	    80: //Error Reading Access
	        #Done := true;
	        #Busy := false;
	        #Error := TRUE;
	        #ErrorId := #st_StatusRead;
	        
	    90:  // Error while Write Access
	        #Done := true;
	        #Busy := false;
	        #Error := TRUE;
	        #ErrorId := #st_StatusWR;
	        
	        
	    100: // read successfully
	        #Done := true;
	        #Busy := false;
	        #Error := false;
	        
	    150:// write successfully
	        #Done := true;
	        #Busy := false;
	        #Error := false;
	        
	    200:  //Error while reading
	        #Done := true;
	        #Busy := false;
	        #Error := TRUE;
	        
	    300:  //Error while writing
	        #Done := true;
	        #Busy := false;
	        #Error := TRUE;
	        
	END_CASE;
	
	IF NOT #Enable THEN
	    #st_step := 0;
	    #st_ReqRef := 1;
	    #Done := false;
	    #Busy := false;
	    #Error := false;
	    #ErrorId := 16#00000000;
	    #ValueReadBOOL := false;
	    #ValueReadLINT := 0;
	    #ValueReadREAL := 0.0;
	    #st_StatusRead := 0;
	    #st_ErrorCounter := 0;
	END_IF;
END_FUNCTION_BLOCK

FUNCTION "Festo_Messages_Drives_EN" : Void
TITLE = Meldungen von CMMT MotorControllern
{ S7_Optimized_Access := 'TRUE' }
AUTHOR : LWNR
VERSION : 1.1
//Dieser Baustein gibt anhand der Meldungs-ID den Meldetext des Diagnose-
//ereignisses in Klartext (als STRING) aus.
//Weiterhin wird die Hauptgruppe, die Untergruppe, die Beschreibung sowie eine Abhilfe der anstehende Diasgnosemeldung in Klartext (als STRING) ausgegeben.
//Es sind alle Arten von Meldungen (Informationen, Warnungen und Fehler) der Geräte CMMT-AS und CMMT-ST enthalten.
   VAR_INPUT 
      ActFault_Drive : Word;   // Actual fault number of the drive
      ActWarning_Drive : Word;   // Actual warning number of the drive
   END_VAR

   VAR_OUTPUT 
      strMessage : String;   // Error or warning message
   END_VAR

   VAR_TEMP 
      MessageNo : Word;
   END_VAR


BEGIN
	(*############################################################
	    FESTO SE & Co. KG, Esslingen
	    Copyright (c) 2020. All rights reserved.    
	
	    NAME OF FUNCTION BLOCK:         Festo_Messages_Drives_EN
	    VERSION NUMBER:                 V1.1
	    COMPOSER:                       Festo
	    
	    -----------------------------------------------------
	   Date        Name                Activity                                                                              
	   20.02.2020  lwnr                created (V1.0)
	   09.12.2022  bkle                name changed 
	                                   Input: ActWarning_Drive added for warnings (V1.1)
	############################################################*)
	IF #ActFault_Drive <> 0 THEN
	    #MessageNo := #ActFault_Drive;
	ELSIF #ActWarning_Drive <> 0 THEN
	    #MessageNo := #ActWarning_Drive;
	END_IF;
	
	CASE WORD_TO_INT(#MessageNo) OF
	    0:
	        #strMessage := 'no error';
	        
	        (***************************************************************************)
	        (*                       Main group 1 - Current                             *)
	        (***************************************************************************)
	        
	        (* Subgroup 1 - Short circuit *)
	    10:
	        #strMessage := 'Short circuit motor phases/braking resistor';
	       
	    11:
	        #strMessage := 'Error on over-current monitoring';
	        
	        
	        (* Subgroup 2 - I²T *)
	    12:
	        #strMessage := 'I2t monitoring: motor warning limit';
	        
	    13:
	        #strMessage := 'I2t monitoring: motor error limit';
	        
	    14:
	        #strMessage := 'I2t monitoring: output stage warning limit';
	
	        
	    15:
	        #strMessage := 'I2t monitoring: output stage error limit';
	        
	    16:
	        #strMessage := 'I2t monitoring: output stage in standstill warning limit';
	        
	    17:
	        #strMessage := 'I2t monitoring: output stage in standstill error limit';
	        
	    18:
	        #strMessage := 'I2t monitoring motor: parameterisation invalid';
	        
	    258:
	        #strMessage := 'I2t monitoring: motor warning limit';
	        
	    259:
	        #strMessage := 'I2t monitoring: motor error limit';
	        
	        (* Subgroup 3 - braking resistor *)
	    19:
	        #strMessage := 'Warning: pulse energy monitoring, braking resistor';
	        
	    20:
	        #strMessage := 'Error: pulse energy monitoring, braking resistor';
	        
	    21:
	        #strMessage := 'Parameterisation of pulse energy monitoring for braking resistor invalid';
	        
	        
	        
	        (***************************************************************************)
	        (*                       Main group 2 - Voltage                          *)
	        (***************************************************************************)
	        
	        (* Subgroup 1 - Supply *)
	    22:
	        #strMessage := 'Undervoltage in logic supply (PS) 24 V DC';
	        
	    23:
	        #strMessage := 'Overvoltage in logic supply (PS) 24 V DC';
	        
	    24:
	        #strMessage := 'Undervoltage in logic supply 5V internal';
	        
	    25:
	        #strMessage := 'Overvoltage in logic supply 5V internal';
	        
	    26:
	        #strMessage := 'Undervoltage in logic supply 3.3V internal';
	        
	    27:
	        #strMessage := 'Overvoltage in logic supply 3.3V internal';
	        
	    28:
	        #strMessage := 'Undervoltage in logic supply safety section 3.3V internal';
	        
	    29:
	        #strMessage := 'Overvoltage in logic supply safety section 3.3V internal';
	        
	        
	        (* Subgroup 2 - intermediate circuit *)
	    30:
	        #strMessage := 'Overvoltage in intermediate circuit';
	        
	    31:
	        #strMessage := 'Undervoltage in intermediate circuit';
	        
	    32:
	        #strMessage := 'Intermediate circuit danger threshold reached';
	        
	    33:
	        #strMessage := 'DC link voltage too low following power failure';
	        
	    34:
	        #strMessage := 'Intermediate circuit precharge time exceeded';
	        
	    35:
	        #strMessage := 'Residual voltage too high following rapid discharge';
	        
	    286:
	        #strMessage := 'The DC relay for loading the DC link does not open';
	        
	    287:
	        #strMessage := 'The DC relay for charging the DC link does not close';
	        
	        
	        (* Subgroup 3 - Mains volatge *)
	    36:
	        #strMessage := 'No mains voltage';
	        
	    37:
	        #strMessage := 'System voltage dip detected';
	        
	    38:
	        #strMessage := 'Undervoltage in power supply';
	        
	    39:
	        #strMessage := 'Overvoltage in power supply';
	        
	    40:
	        #strMessage := 'Phase failure in power supply';
	        
	    41:
	        #strMessage := 'Powersupply signal shape NOT as configured';
	        
	    251:
	        #strMessage := 'Deactivation threshold for energy recovery reached';
	        
	        
	        
	        (* Subgroup 4 - Encoder supply voltage *)
	    42:
	        #strMessage := 'Supply voltage for encoder is outside monitoring thresholds';
	        
	    43:
	        #strMessage := 'Encoder supply voltage control failed';
	        
	        
	        (***************************************************************************)
	        (*                     Main group 3 - TEMPERATURE                          *)
	        (***************************************************************************)
	        
	        (* Subgroup 1 - GERAET *)
	    44:
	        #strMessage := 'Warning threshold: Insufficient temperature in device';
	        
	    45:
	        #strMessage := 'Insufficient temperature in device';
	        
	    46:
	        #strMessage := 'Warning threshold: Device overtemperature';
	        
	    47:
	        #strMessage := 'Device overtemperature';
	        
	        
	        (* Subgroup 2 - Output stage *)
	    48:
	        #strMessage := 'Warning threshold: Insufficient temperature in power section';
	        
	    49:
	        #strMessage := 'Insufficient temperature in output stage';
	        
	    50:
	        #strMessage := 'Warning threshold: Power section overtemperature';
	        
	    51:
	        #strMessage := 'Power section overtemperature';
	        
	        
	        (* Subgroup 3 - MOTOR *)
	    52:
	        #strMessage := 'Warning threshold: Insufficient temperature in motor';
	        
	    53:
	        #strMessage := 'Insufficient temperature in motor';
	        
	    54:
	        #strMessage := 'Warning threshold: Motor overtemperature';
	        
	    55:
	        #strMessage := 'Motor overtemperature';
	        
	        
	        (***************************************************************************)
	        (*                       Main group 5 - Motion                          *)
	        (***************************************************************************)
	        
	        (* Subgroup 1 - Homing *)
	    56:
	        #strMessage := 'Parameterisation of homing run invalid';
	        
	    57:
	        #strMessage := 'Homing: Timeout';
	        
	    58:
	        #strMessage := 'Homing: Search path exceeded';
	        
	        
	        (* Subgroup 2 - Movement calculation *)
	    59:
	        #strMessage := 'Task invalid';
	        
	    60:
	        #strMessage := 'Unknown motion task pending';
	        
	    61:
	        #strMessage := 'Task could not be executed as the drive control is missing';
	        
	    62:
	        #strMessage := 'Task could not be executed as a safety function is requested';
	        
	    63:
	        #strMessage := 'Calculation of brake travel failed';
	        
	    64:
	        #strMessage := 'Task could not be executed as no DC link voltage is present';
	        
	    65:
	        #strMessage := 'Motion task rejected in current status';
	        
	    66:
	        #strMessage := 'Task could not be executed as the encoder is not ready';
	        
	    67:
	        #strMessage := 'Task could not be executed as the drive is not referenced';
	        
	    68:
	        #strMessage := 'Task could not be executed as a reinitialization is required due to a parameter change';
	        
	    69:
	        #strMessage := 'Task could not be executed as a restart is required due to a parameter change';
	        
	    71:
	        #strMessage := 'An error occurred in the trajectory generator when calculating a movement profile';
	        
	    72:
	        #strMessage := 'The position specified for the trajectory generator is invalid';
	        
	    73:
	        #strMessage := 'The speed specified for the trajectory generator is invalid';
	        
	    74:
	        #strMessage := 'The acceleration specified for the trajectory generator is invalid';
	        
	    75:
	        #strMessage := 'The delay specified for the trajectory generator is invalid';
	        
	    76:
	        #strMessage := 'The jerk specified for the trajectory generator is invalid';
	        
	    77:
	        #strMessage := 'An error occurred in the trajectory generator when calculating a movement profile';
	        
	    78:
	        #strMessage := 'Stop ramp: Timeout';
	        
	    79:
	        #strMessage := 'The torque increase is invalid';
	        
	    80:
	        #strMessage := 'Simultaneous negative/positive directional lock';
	        
	    245:
	        #strMessage := 'Received PDO outside tolerance window';
	        
	    278:
	        #strMessage := 'Order could not be executed because a directional lock is active';
	        
	    279:
	        #strMessage := 'Fixed stop not reached';
	        
	    280:
	        #strMessage := 'Monitoring window exit fixed stop';
	        
	    364:
	        #strMessage := 'The preset profile velocity is 0';
	        
	        (***************************************************************************)
	        (*             Main group 6 - KONFIGURATION                *)
	        (***************************************************************************)
	        
	        (* Subgroup 0 - no categorie *)
	    70:
	        #strMessage := 'Record table parameter is invalid';
	        
	    81:
	        #strMessage := 'The operating mode of the regulator (position, speed, force, stop) does not match the parameterisation';
	        
	    82:
	        #strMessage := 'The parameterisation of the notch filter frequency is invalid';
	        
	    83:
	        #strMessage := 'Record table incorrect';
	        
	    84:
	        #strMessage := 'Parameterisation of switching frequency invalid';
	        
	    85:
	        #strMessage := 'The configuration of the digital inputs or outputs is invalid';
	        
	    248:
	        #strMessage := 'The parameterized motor type (servo, stepper, ...) is not supported';
	        
	    252:
	        #strMessage := 'Start and end voltage for reactive current braking incompatible';
	        
	    313:
	        #strMessage := 'Selection data trigger in function Variable signalling function invalid';
	        
	        
	        (* Subgroup 2 - Boundary value *)
	    86:
	        #strMessage := 'Setpoint torque and speed limit do not match';
	        
	    87:
	        #strMessage := 'Speed control limitation invalid';
	        
	    88:
	        #strMessage := 'Torque control limitation invalid';
	        
	    89:
	        #strMessage := 'Current control limitation invalid';
	        
	    90:
	        #strMessage := 'Maximum peak current control limitation invalid';
	        
	    91:
	        #strMessage := 'Parameterisation of nominal current/maximum peak current of motor invalid';
	        
	    273:
	        #strMessage := 'Change of control mode not permitted';
	        
	    274:
	        #strMessage := 'Movement order not permitted in controlled operation';
	        
	    275:
	        #strMessage := 'Change to close-loop operation not permitted';
	        
	        
	        (* Subgroup 5 - Parameter set *)
	    97:
	        #strMessage := 'Parameter set not found';
	        
	    98:
	        #strMessage := 'Parameter set invalid';
	        
	    99:
	        #strMessage := 'Parameter set incompatible';
	        
	    100:
	        #strMessage := 'Parameter not found';
	        
	    101:
	        #strMessage := 'Parameter not writable';
	        
	    102:
	        #strMessage := 'Transmission error in parameter set';
	        
	    103:
	        #strMessage := 'Parameter set: store failed';
	        
	    104:
	        #strMessage := 'Parameter set: delete failed';
	        
	    105:
	        #strMessage := 'Factory parameter not found';
	        
	    106:
	        #strMessage := 'Factory parameter set invalid';
	        
	    107:
	        #strMessage := 'Factory parameter set not found';
	        
	    108:
	        #strMessage := 'Factory parameter set incompatible';
	        
	    290:
	        #strMessage := 'Parameter set version older';
	        
	    291:
	        #strMessage := 'Parameter set version newer';
	        
	        
	        (***************************************************************************)
	        (*                        Main group 7 - Monitoring                      *)
	        (***************************************************************************)
	        
	        (* Subgroup 1 - Limits *)
	    109:
	        #strMessage := 'Negative software end position';
	        
	    110:
	        #strMessage := 'Positive software end position';
	        
	    111:
	        #strMessage := 'Limitation negative direction';
	        
	    112:
	        #strMessage := 'Limitation positive direction';
	        
	    113:
	        #strMessage := 'Parameterisation of software end positions';
	        
	    114:
	        #strMessage := 'Negative hardware limit switch reached';
	        
	    115:
	        #strMessage := 'Positive hardware limit switch reached';
	        
	    116:
	        #strMessage := 'Limitation by negative hardware limit switch';
	        
	    117:
	        #strMessage := 'Limitation by positive hardware limit switch';
	        
	    118:
	        #strMessage := 'Error: both hardware limit switches occupied';
	        
	    119:
	        #strMessage := 'Negative stroke limit reached';
	        
	    120:
	        #strMessage := 'Positive stroke limit reached';
	        
	        
	        (* Subgroup 2 - Motion monitoring *)
	    121:
	        #strMessage := 'Target position reached';
	        
	    122:
	        #strMessage := 'Target speed reached';
	        
	    123:
	        #strMessage := 'Target torque reached';
	        
	    124:
	        #strMessage := 'Standstill reached';
	        
	    125:
	        #strMessage := 'Standstill reached and within standstill window';
	        
	    126:
	        #strMessage := 'Position error: following error';
	        
	    127:
	        #strMessage := 'velocity: following error';
	        
	    128:
	        #strMessage := 'velocity monitoring reports velocity too high';
	        
	    129:
	        #strMessage := 'Drive has left the target range';
	        
	    130:
	        #strMessage := 'Reverse feed monitoring reports error';
	        
	    131:
	        #strMessage := 'Residual distance too low';
	        
	    132:
	        #strMessage := 'Trajectory completed setpoint value reached';
	        
	    133:
	        #strMessage := 'Position difference encoder 1 to encoder 2 too large';
	        
	        
	        (* Subgroup 3 - boundary values *)
	    134:
	        #strMessage := 'Voltage limiting active';
	        
	    135:
	        #strMessage := 'A limit for the speed or current is active';
	        
	        
	        (* Subgroup 4 - Zero angle *)
	    136:
	        #strMessage := 'Zero-angle location failed';
	        
	    137:
	        #strMessage := 'Commutation finding error';
	        
	        
	        (* Subgroup 5 - analog input *)
	    138:
	        #strMessage := 'Analogue setpoint specification limit exceeded';
	        
	        
	        
	        (***************************************************************************)
	        (*                      Main group 8 - Communication                       *)
	        (***************************************************************************)
	        
	        (* Subgroup 0 - no categorie *)
	    139:
	        #strMessage := 'Fieldbus not supported';
	        
	    140:
	        #strMessage := 'Failure of fieldbus synchronisation signal';
	        
	    243:
	        #strMessage := 'Invalid cycle time';
	        
	        
	        (* Subgroup 3 - PROFINET *)
	    141:
	        #strMessage := 'Invalid process data';
	        
	    373:
	        #strMessage := 'Failure of communication processor synchronisation';
	        
	        
	        (* Subgroup 9 - PROFIDRIVE *)
	    144:
	        #strMessage := 'Application class not supported';
	        
	    145:
	        #strMessage := 'Telegram not supported';
	        
	    288:
	        #strMessage := 'ProfiDrive test fault 1';
	        
	    289:
	        #strMessage := 'ProfiDrive test fault 2';
	        
	    294:
	        #strMessage := 'PLC Control Bit is not set';
	        
	    299:
	        #strMessage := 'clock cycle synchronous operation sign-of-life failure';
	        
	    382:
	        #strMessage := 'Invalid configuration Extended process data';
	        
	        
	        (* Subgroup 12 - others *)
	    250:
	        #strMessage := 'Invalid operating mode';
	        
	    272:
	        #strMessage := 'Resolution position factor group invalid';
	        
	        
	        (***************************************************************************)
	        (*                     Main group 9 - Safety                               *)
	        (***************************************************************************)
	        
	        (* Subgroup 0 - no categorie *)
	    146:
	        #strMessage := 'Safety function requested';
	        
	    147:
	        #strMessage := 'Plausibility check of safety feedback signals';
	        
	        
	        (* Subgroup 1 - STO *)
	    148:
	        #strMessage := 'STO: Discrepancy time exceeded';
	        
	    149:
	        #strMessage := 'Plausibility check #STO-A/B';
	        
	    150:
	        #strMessage := 'Sequence monitoring #STO-A/B';
	        
	        
	        (* Subgroup 2 - SBC *)
	    151:
	        #strMessage := 'Plausibility check #SBC-A/B';
	        
	    152:
	        #strMessage := 'SBC: Discrepancy time exceeded';
	        
	        
	        (***************************************************************************)
	        (*                     Main group 10 - Internal hardware                   *)
	        (***************************************************************************)
	        
	        (* Subgroup 1 - Module error *)
	    153:
	        #strMessage := 'RTE module cannot be reached';
	        
	    154:
	        #strMessage := 'Internalisation of RTE module failed';
	        
	    155:
	        #strMessage := 'Error: fan faulty';
	        
	    156:
	        #strMessage := 'Common error power output stage';
	        
	    157:
	        #strMessage := 'FPGA does not start up';
	        
	    158:
	        #strMessage := 'FPGA version invalid';
	        
	    199:
	        #strMessage := 'Synchronisation with FPGA failed';
	        
	    249:
	        #strMessage := 'Error RTE module watchdog monitoring';
	        
	        
	        
	        (***************************************************************************)
	        (*                         Main group 11 - SOFTWARE                       *)
	        (***************************************************************************)
	        
	        (* Subgroup 1 - EXCEPTION *)
	        
	    159:
	        #strMessage := 'Data directory memory full';
	        
	    160:
	        #strMessage := 'Data directory indexed twice';
	        
	    161:
	        #strMessage := 'Overflow diagnostic register';
	        
	    162:
	        #strMessage := 'Overflow diagnostic register buffer';
	        
	    163:
	        #strMessage := 'Error user unit conversion';
	        
	    244:
	        #strMessage := 'Undervoltage RTE module';
	        
	        
	        (* Subgroup 2 - TASK *)
	    164:
	        #strMessage := 'Process runtime exceeded';
	        
	    165:
	        #strMessage := 'Timeout process level 0';
	        
	    166:
	        #strMessage := 'Timeout process level 1';
	        
	    167:
	        #strMessage := 'Timeout process level 2';
	        
	    168:
	        #strMessage := 'Timeout process level 3';
	        
	    169:
	        #strMessage := 'Timeout process level 4';
	        
	    170:
	        #strMessage := 'Timeout process level 5';
	        
	    171:
	        #strMessage := 'Timeout process level 6';
	        
	    172:
	        #strMessage := 'Timeout process level 7';
	        
	        
	        (* Subgroup 3 - File system *)
	    173:
	        #strMessage := 'File system faulty';
	        
	    174:
	        #strMessage := 'File: user file (backup) invalid';
	        
	    175:
	        #strMessage := 'Creation of user file (backup) not possible';
	        
	    176:
	        #strMessage := 'CRC error in user file';
	        
	    177:
	        #strMessage := 'File: user file invalid';
	        
	    178:
	        #strMessage := 'New user file has been created';
	        
	    179:
	        #strMessage := 'Writing to user file not possible';
	        
	    180:
	        #strMessage := 'Unknown user file error';
	        
	        
	        (* Subgroup 4 - FIRMWAREUPDATE *)
	    181:
	        #strMessage := 'Writing to firmware failed';
	        
	    182:
	        #strMessage := 'Reading from firmware failed';
	        
	    183:
	        #strMessage := 'Firmware invalid';
	        
	    184:
	        #strMessage := 'Firmware incompatible';
	        
	    185:
	        #strMessage := 'Firmware save location invalid';
	        
	    186:
	        #strMessage := 'Firmware save location empty';
	        
	    187:
	        #strMessage := 'Firmware update not allowed';
	        
	    188:
	        #strMessage := 'Firmware package in use';
	        
	    189:
	        #strMessage := 'System error during firmware update';
	        
	    190:
	        #strMessage := 'Firmware update failed';
	        
	        
	        (* Subgroup 5 - Device configuration *)
	    191:
	        #strMessage := 'Calibration data incorrect: Safety';
	        
	    192:
	        #strMessage := 'Device data incorrect';
	        
	    193:
	        #strMessage := 'Device data incorrect: control section';
	        
	    194:
	        #strMessage := 'Device data incorrect: communication section';
	        
	    195:
	        #strMessage := 'Device data incorrect: Safety';
	        
	    196:
	        #strMessage := 'Calibration data incorrect: control section';
	        
	    197:
	        #strMessage := 'Calibration data incorrect: power section';
	        
	    198:
	        #strMessage := 'Device data incorrect: power section';
	        
	    200:
	        #strMessage := 'Current sensor calibration invalid';
	        
	    201:
	        #strMessage := 'Device not configured';
	        
	    202:
	        #strMessage := 'Device data: store failed';
	        
	        
	        (* Subgroup 6 - LIBRTE *)
	    203:
	        #strMessage := 'Answer to a read request missing in LibRTE';
	        
	    285:
	        #strMessage := 'Error communication module mailbox';
	        
	    300:
	        #strMessage := 'COM module error';
	        
	        
	        (* Subgroup 7 - WARMSTART *)
	    204:
	        #strMessage := 'Initialization failed';
	        
	    205:
	        #strMessage := 'Task ignored as reinitialization not possible';
	        
	    271:
	        #strMessage := 'Reinitialization failed';
	        
	        
	        (* Subgroup 8 - version  management *)
	    206:
	        #strMessage := 'Hardware does not correspond to expected revision status';
	        
	    207:
	        #strMessage := 'Hardware does not correspond to expected compatibility state';
	        
	        
	        
	        (***************************************************************************)
	        (*                         Main group 12 - maintenance                        *)
	        (***************************************************************************)
	        
	        (* Subgroup 1 - Mileage *)
	    208:
	        #strMessage := 'Maximum value for the mileage is reached';
	        
	    209:
	        #strMessage := 'Mileage danger threshold reached';
	        
	    210:
	        #strMessage := 'Mileage error threshold reached';
	        
	    211:
	        #strMessage := 'Maximum load change value reached';
	        
	    212:
	        #strMessage := 'Load change danger threshold reached';
	        
	    213:
	        #strMessage := 'Load change error threshold reached';
	        
	        
	        
	        (***************************************************************************)
	        (*                      Main group 13 - Others                     *)
	        (***************************************************************************)
	        
	        (* Subgroup 1 - diagnosis *)
	    214:
	        #strMessage := 'Message acknowledgment';
	        
	    215:
	        #strMessage := 'Diagnostics log file has invalid format';
	        
	    216:
	        #strMessage := 'Loss of messages from diagnostics log';
	        
	        
	        (* Subgroup 2 - AUTOTUNING *)
	    217:
	        #strMessage := 'Autotuning aborted';
	        
	    218:
	        #strMessage := 'Autotuning travel insufficient';
	        
	    219:
	        #strMessage := 'Autotuning controller parameters invalid';
	        
	    220:
	        #strMessage := 'Transmission of autotuning measured values failed';
	        
	        
	        
	        
	        
	        
	        (***************************************************************************)
	        (*                     Main group 16 - External device                     *)
	        (***************************************************************************)
	        
	        (* Subgroup 1 - CDSB *)
	    221:
	        #strMessage := 'CDSB display file faulty';
	        
	    222:
	        #strMessage := 'JSON display description for CDSB too large';
	        
	    223:
	        #strMessage := 'SPI communication too slow';
	        
	        
	        
	        
	        
	        (***************************************************************************)
	        (*                   Main group 17 - Safety (data)                         *)
	        (***************************************************************************)
	        
	        (* Subgroup 1 - User login *)
	    224..225:
	        #strMessage := 'Login completed';
	        
	    226:
	        #strMessage := 'Login error';
	        
	        
	        
	        
	        
	        (***************************************************************************)
	        (*                        Main group 18 - Encoder                          *)
	        (***************************************************************************)
	        
	        (* Subgroup 0 - no cetegorie *)
	    92:
	        #strMessage := 'Motor change detected, commutation angle invalid';
	        
	    93:
	        #strMessage := 'Motor change detected, zero point offset invalid';
	        
	    94:
	        #strMessage := 'Commutation angle in encoder invalid';
	        
	    95:
	        #strMessage := 'Encoder type plate invalid';
	        
	    96:
	        #strMessage := 'Encoder type plate (user-defined) invalid';
	        
	    227:
	        #strMessage := 'Encoder identification reports incorrect encoder type';
	        
	    318:
	        #strMessage := 'State transition error';
	        
	        
	        (* Subgroup 1 - ENDAT*)
	    228:
	        #strMessage := 'Common error EnDat 2.1';
	        
	    229:
	        #strMessage := 'Common error EnDat 2.2';
	        
	        
	        (* Subgroup 2 - HYPERFACE*)
	    230:
	        #strMessage := 'Vector length invalid';
	        
	    231:
	        #strMessage := 'Quadrant invalid';
	        
	    232:
	        #strMessage := 'Hiperface communication timeout';
	        
	    233:
	        #strMessage := 'Error in CRC protocol Hiperface';
	        
	    234:
	        #strMessage := 'Common error Hiperface';
	        
	    276:
	        #strMessage := 'Quadrant unstable';
	        
	        
	        (* Subgroup 3 - QUADRATURE (incremental encoder)*)
	    235:
	        #strMessage := 'Incremental encoder analysis invalid';
	        
	    301:
	        #strMessage := 'Increments between Z-pulses invalid';
	        
	        
	        (* Subgroup 4 - NIKON A*)
	    236:
	        #strMessage := 'Protocol error Nikon-A encoder';
	        
	    237:
	        #strMessage := 'Timeout Nikon-A encoder';
	        
	    238:
	        #strMessage := 'CRC error Nikon-A encoder';
	        
	        
	        (* Subgroup 5 - BISS C*)
	    239:
	        #strMessage := 'BISSC encoder analysis invalid';
	        
	        
	        (* Subgroup 6 - SIN/COS*)
	    240:
	        #strMessage := 'Vector length invalid';
	        
	    241:
	        #strMessage := 'Quadrant invalid';
	        
	    242:
	        #strMessage := 'Timeout Geberinitialisierung';
	        
	    277:
	        #strMessage := 'Error SIN/COS-encoder';
	        
	        
	        (* Subgroup 7 - encoder systems *)
	    365:
	        #strMessage := 'Invalid request Gn_STW1.4...7';
	        
	    366:
	        #strMessage := 'Function not supported Gn_STW1';
	        
	    367:
	        #strMessage := 'Axis parking not possible';
	        
	    368:
	        #strMessage := 'Error reference marks search';
	        
	    369:
	        #strMessage := 'Error Read Position Reference mark';
	        
	    370:
	        #strMessage := 'Error measuring on the fly';
	        
	    371:
	        #strMessage := 'Error Read Position Measure on the fly';
	        
	    372:
	        #strMessage := 'Error Transfer absolute position to Gn_XIST2';
	        
	    ELSE  // Statement section ELSE
	        #strMessage := 'unknown';
	END_CASE;
	
END_FUNCTION

FUNCTION_BLOCK "LK_G5000"   // FB6, LAD
{ S7_Optimized_Access := 'TRUE' }
VERSION : 0.1
// stored: AutoNumber true, IsIECCheckEnabled false, IsRetainMemResEnabled false, MemoryReserve 100, SetENOAutomatically false, UDAEnableTagReadback false
BEGIN

REGION Network 1: Write / Read data in and from DB - CTRL_ BITS
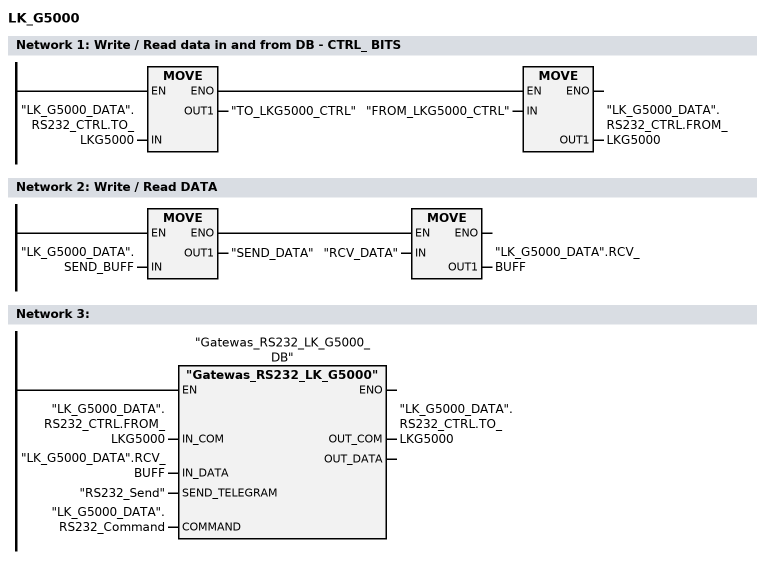
   RUNG wire#powerrail
      Move(in := "LK_G5000_DATA".RS232_CTRL.TO_LKG5000, out1 => "TO_LKG5000_CTRL")
      Move(in := "FROM_LKG5000_CTRL", out1 => "LK_G5000_DATA".RS232_CTRL.FROM_LKG5000)
   END_RUNG
   // the same network as SCL:
   "TO_LKG5000_CTRL" := "LK_G5000_DATA".RS232_CTRL.TO_LKG5000;
   "LK_G5000_DATA".RS232_CTRL.FROM_LKG5000 := "FROM_LKG5000_CTRL";
END_REGION

REGION Network 2: Write / Read DATA
   RUNG wire#powerrail
      Move(in := "LK_G5000_DATA".SEND_BUFF, out1 => "SEND_DATA")
      Move(in := "RCV_DATA", out1 => "LK_G5000_DATA".RCV_BUFF)
   END_RUNG
   // the same network as SCL:
   "SEND_DATA" := "LK_G5000_DATA".SEND_BUFF;
   "LK_G5000_DATA".RCV_BUFF := "RCV_DATA";
END_REGION

REGION Network 3
   RUNG wire#powerrail
      "Gatewas_RS232_LK_G5000_DB"(IN_COM := "LK_G5000_DATA".RS232_CTRL.FROM_LKG5000, IN_DATA := "LK_G5000_DATA".RCV_BUFF, SEND_TELEGRAM := "RS232_Send", COMMAND := "LK_G5000_DATA".RS232_Command, OUT_COM => "LK_G5000_DATA".RS232_CTRL.TO_LKG5000, OUT_DATA =>)
   END_RUNG
   // the same network as SCL:
   "Gatewas_RS232_LK_G5000_DB"(IN_COM := "LK_G5000_DATA".RS232_CTRL.FROM_LKG5000,   // "Gatewas_RS232_LK_G5000"
                           IN_DATA := "LK_G5000_DATA".RCV_BUFF,
                           SEND_TELEGRAM := "RS232_Send",
                           COMMAND := "LK_G5000_DATA".RS232_Command,
                           OUT_COM => "LK_G5000_DATA".RS232_CTRL.TO_LKG5000);
END_REGION
END_FUNCTION_BLOCK

FUNCTION_BLOCK "Gatewas_RS232_LK_G5000"   // FB10, LAD
{ S7_Optimized_Access := 'TRUE' }
VERSION : 0.1
// stored: AutoNumber true, IsIECCheckEnabled false, IsRetainMemResEnabled false, MemoryReserve 100, SetENOAutomatically false, UDAEnableTagReadback false
   VAR_INPUT
      IN_COM : "UDT_LKG5000_RS232_RCV";
      IN_DATA : "UDT_RS232_RCV_DATA";
      SEND_TELEGRAM : Bool;
      COMMAND : String[10];
   END_VAR
   VAR_OUTPUT
      OUT_COM : "UDT_LKG5000_RS232_SEND";
      OUT_DATA : "UDT_RS232_SEND_DATA";
   END_VAR
   VAR
      COMMAND_SIGN : Array[0..10] of Char;
      Cnt_Command : UInt;
      IEC_Timer_0_Instance { S7_SetPoint := 'True'} : TOF_TIME;
      IEC_Timer_0_Instance_1 { S7_SetPoint := 'True'} : TOF_TIME;
   END_VAR
BEGIN

REGION Network 2 (SCL)
   Strg_TO_Chars(Strg:=#COMMAND,
                 pChars:=0,
                 Cnt=>#Cnt_Command,
                 Chars:=#COMMAND_SIGN);





   // Send frame
   #OUT_COM.Sendframe_size := 20;
   // Receive Frame
   #OUT_COM.Recvframe_size := 20;


   //#OUT_DATA.Data[0] := B#16#02;
   #OUT_DATA.Data[0] := #COMMAND_SIGN[0];
   #OUT_DATA.Data[1] := #COMMAND_SIGN[1];
   #OUT_DATA.Data[2] := #COMMAND_SIGN[2];
   #OUT_DATA.Data[3] := #COMMAND_SIGN[3];
   #OUT_DATA.Data[4] := #COMMAND_SIGN[4];
   #OUT_DATA.Data[5] :=  B#16#D0;

   //#OUT_DATA.Data[5] := #COMMAND_SIGN[5];
   //#OUT_DATA.Data[6] := #COMMAND_SIGN[6];
   //#OUT_DATA.Data[7] := #COMMAND_SIGN[7];
   //#OUT_DATA.Data[8] := #COMMAND_SIGN[8];
   //#OUT_DATA.Data[9] := #COMMAND_SIGN[9];
   //#OUT_DATA.Data[10] := #COMMAND_SIGN[10];
   //#OUT_DATA.Data[11] := #COMMAND_SIGN[11];
   //#OUT_DATA.Data[12] := #COMMAND_SIGN[12];
   //#OUT_DATA.Data[13] := #COMMAND_SIGN[13];
   //#OUT_DATA.Data[14] := #COMMAND_SIGN[14];
   //#OUT_DATA.Data[15] := #COMMAND_SIGN[15];
   //#OUT_DATA.Data[16] := #COMMAND_SIGN[16];
   //#OUT_DATA.Data[17] := #COMMAND_SIGN[17];
   //#OUT_DATA.Data[18] := #COMMAND_SIGN[18];
   //#OUT_DATA.Data[19] := #COMMAND_SIGN[19];
   //#OUT_DATA.Data[20] := #COMMAND_SIGN[20];
   //#OUT_DATA.Data[21] := #COMMAND_SIGN[21];
   //#OUT_DATA.Data[22] := #COMMAND_SIGN[22];
   //#OUT_DATA.Data[23] := B#16#D0;


   "R_TRIG_DB"(CLK:=#SEND_TELEGRAM);

   "IEC_Timer_0_DB".TP(IN:="R_TRIG_DB".Q,
                       PT:=T#2s);

   #OUT_COM.CTRL_Send := "IEC_Timer_0_DB".Q;


   "F_TRIG_DB"(CLK:=#OUT_COM.CTRL_Send);
END_REGION

REGION Network 3
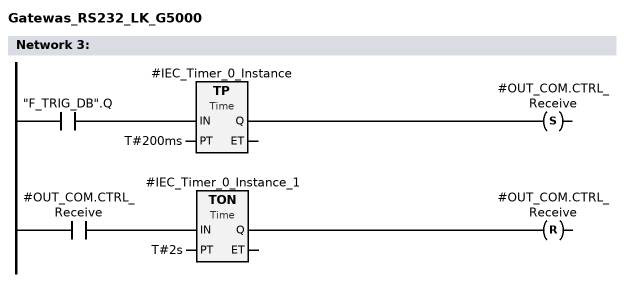
   RUNG wire#powerrail
      Contact( "F_TRIG_DB".Q )
      { S7_Templates := "time_type := Time" } #IEC_Timer_0_Instance.TP(pt := T#200ms, et =>)
      S_Coil( #OUT_COM.CTRL_Receive )
   END_RUNG
   RUNG wire#powerrail
      Contact( #OUT_COM.CTRL_Receive )
      { S7_Templates := "time_type := Time" } #IEC_Timer_0_Instance_1.TON(pt := T#2s, et =>)
      R_Coil( #OUT_COM.CTRL_Receive )
   END_RUNG
   // the same network as SCL:
   #IEC_Timer_0_Instance(IN := "F_TRIG_DB".Q, PT := T#200ms);   // TP
   IF #IEC_Timer_0_Instance.Q THEN #OUT_COM.CTRL_Receive := TRUE; END_IF;
   #IEC_Timer_0_Instance_1(IN := #OUT_COM.CTRL_Receive, PT := T#2s);   // TON
   IF #IEC_Timer_0_Instance_1.Q THEN #OUT_COM.CTRL_Receive := FALSE; END_IF;
END_REGION
END_FUNCTION_BLOCK

FUNCTION_BLOCK "FB_LJ_X8000"   // FB11, LAD
{ S7_Optimized_Access := 'TRUE' }
VERSION : 0.1
// stored: AutoNumber true, IsIECCheckEnabled false, IsRetainMemResEnabled false, MemoryReserve 100, SetENOAutomatically false, UDAEnableTagReadback false
BEGIN

REGION Network 1: 02_LJ_X8000_Control
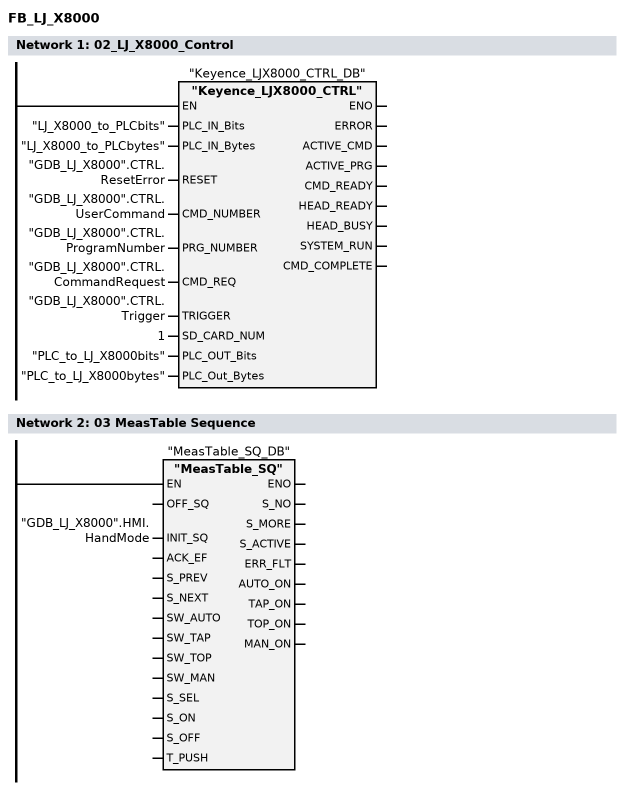
   RUNG wire#powerrail
      "Keyence_LJX8000_CTRL_DB"(PLC_IN_Bits := "LJ_X8000_to_PLCbits", PLC_IN_Bytes := "LJ_X8000_to_PLCbytes", RESET := "GDB_LJ_X8000".CTRL.ResetError, CMD_NUMBER := "GDB_LJ_X8000".CTRL.UserCommand, PRG_NUMBER := "GDB_LJ_X8000".CTRL.ProgramNumber, CMD_REQ := "GDB_LJ_X8000".CTRL.CommandRequest, TRIGGER := "GDB_LJ_X8000".CTRL.Trigger, SD_CARD_NUM := 1, PLC_OUT_Bits := "PLC_to_LJ_X8000bits", PLC_Out_Bytes := "PLC_to_LJ_X8000bytes", ERROR =>, ACTIVE_CMD =>, ACTIVE_PRG =>, CMD_READY =>, HEAD_READY =>, HEAD_BUSY =>, SYSTEM_RUN =>, CMD_COMPLETE =>)
   END_RUNG
   // the same network as SCL:
   "Keyence_LJX8000_CTRL_DB"(PLC_IN_Bits := "LJ_X8000_to_PLCbits",   // "Keyence_LJX8000_CTRL"
                           PLC_IN_Bytes := "LJ_X8000_to_PLCbytes",
                           RESET := "GDB_LJ_X8000".CTRL.ResetError,
                           CMD_NUMBER := "GDB_LJ_X8000".CTRL.UserCommand,
                           PRG_NUMBER := "GDB_LJ_X8000".CTRL.ProgramNumber,
                           CMD_REQ := "GDB_LJ_X8000".CTRL.CommandRequest,
                           TRIGGER := "GDB_LJ_X8000".CTRL.Trigger,
                           SD_CARD_NUM := 1,
                           PLC_OUT_Bits := "PLC_to_LJ_X8000bits",
                           PLC_Out_Bytes := "PLC_to_LJ_X8000bytes");
END_REGION

REGION Network 2: 03 MeasTable Sequence
   RUNG wire#powerrail
      "MeasTable_SQ_DB"(OFF_SQ :=, INIT_SQ := "GDB_LJ_X8000".HMI.HandMode, ACK_EF :=, S_PREV :=, S_NEXT :=, SW_AUTO :=, SW_TAP :=, SW_TOP :=, SW_MAN :=, S_SEL :=, S_ON :=, S_OFF :=, T_PUSH :=, S_NO =>, S_MORE =>, S_ACTIVE =>, ERR_FLT =>, AUTO_ON =>, TAP_ON =>, TOP_ON =>, MAN_ON =>)
   END_RUNG
   // the same network as SCL:
   "MeasTable_SQ_DB"(INIT_SQ := "GDB_LJ_X8000".HMI.HandMode);   // "MeasTable_SQ"
END_REGION

REGION Network 3 (SCL): 04 Battery CASE

   "MeasTable_SQ_DB".DataHasRead_1 := FALSE;

   IF "MeasTable_SQ_DB".SQ_ProgramRequest THEN

       CASE "GDB_LJ_X8000".HMI.CellType OF
           1:  // Battery cell 1
               "GDB_LJ_X8000".CTRL.ProgramNumber := 3;
               "DB_CMMT_ST".SetPosition_mm := 650.0;

           2:  // Battey cell 2 
               "GDB_LJ_X8000".CTRL.ProgramNumber := 4;
               "DB_CMMT_ST".SetPosition_mm := 712.0;
           3:  // Battery cell 3
               "GDB_LJ_X8000".CTRL.ProgramNumber := 5;
               "DB_CMMT_ST".SetPosition_mm := 815.0;
           ELSE  // Statement section ELSE
               "DB_CMMT_ST".SetPosition_mm := 240.0;
       END_CASE;

       "MeasTable_SQ_DB".DataHasRead_1 := TRUE;

   END_IF;
END_REGION

REGION Network 4 (SCL): Länge und Breite
   "GDB_LJ_X8000".Cell_MeasData.Länge := "LJ_X8000_to_PLCbytes".T101_DistanceMax / 1000.0;
   "GDB_LJ_X8000".Cell_MeasData.Breite := "LJ_X8000_to_PLCbytes".T101_NoOfNGProfiles / 1000.0;
END_REGION
END_FUNCTION_BLOCK

FUNCTION_BLOCK "Keyence_LJX8000_CTRL"   // FB14, LAD
{ S7_Optimized_Access := 'TRUE' }
VERSION : 0.1
// stored: AutoNumber true, IsIECCheckEnabled false, IsRetainMemResEnabled false, MemoryReserve 100, SetENOAutomatically false, UDAEnableTagReadback false
   VAR_INPUT
      PLC_IN_Bits : "UDT_LJ_X8000 --> PLC_Bits";
      PLC_IN_Bytes : "UDT_LJ_X8000 --> PLC_Bytes";
      RESET : Bool;
      CMD_NUMBER : DInt;
      PRG_NUMBER : DInt;
      CMD_REQ : Bool;
      TRIGGER : Bool;
      SD_CARD_NUM : DInt := 1;
   END_VAR
   VAR_OUTPUT
      ERROR : Bool;
      ACTIVE_CMD : DInt;
      ACTIVE_PRG : DInt;
      CMD_READY : Bool;
      HEAD_READY : Bool;
      HEAD_BUSY : Bool;
      SYSTEM_RUN : Bool;
      CMD_COMPLETE : Bool;
   END_VAR
   VAR_IN_OUT
      PLC_OUT_Bits : "UDT_PLC --> LJ_X8000_Bits";
      PLC_Out_Bytes : "UDT_PLC --> LJ_X8000_Bytes";
   END_VAR
   VAR
      ChangeToRun : Bool;
      ChangeToSetup : Bool;
   END_VAR
   VAR CONSTANT
      T1_Trigger : DInt := 1;
      R0_SwitchToRunMode : DInt := 8;
      S0_SwitchToSetupMode : DInt := 9;
      RS_Reset : DInt := 10;
      RB_Reboot : DInt := 11;
      SS_SaveProgram : DInt := 12;
      CE_ClearError : DInt := 13;
      VW_ChangeTheOperationScreen : DInt := 14;
      RM_ReadRunSetupMode : DInt := 16;
      PW_ChangeInspectionPrograms : DInt := 24;
      PR_ReadProgramSetting : DInt := 25;
      CTD_TriggerDelay : DInt := 34;
   END_VAR
BEGIN

REGION Network 1: Bit0
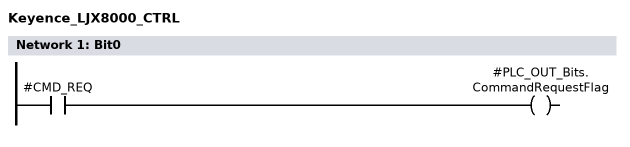
   RUNG wire#powerrail
      Contact( #CMD_REQ )
      Coil( #PLC_OUT_Bits.CommandRequestFlag )
   END_RUNG
   // the same network as SCL:
   #PLC_OUT_Bits.CommandRequestFlag := #CMD_REQ;
END_REGION

REGION Network 2 (SCL): Move data from PLC to Keyence
   #PLC_Out_Bytes.CommandNumber := #CMD_NUMBER;
   #PLC_Out_Bytes.ProgNumber := #PRG_NUMBER;
   #PLC_Out_Bytes.SDCardNumber := #SD_CARD_NUM;


   #PLC_OUT_Bits.ErrorResetRequestFlag := #RESET;
   #PLC_OUT_Bits.Trigger := #TRIGGER;


   #ACTIVE_CMD := #PLC_Out_Bytes.CommandNumber;
END_REGION

REGION Network 3 (SCL): Read data from Keyence
   #ERROR := #PLC_IN_Bits.Error;
   #CMD_READY := #PLC_IN_Bits.CommandReadFlag;
   #HEAD_READY := #PLC_IN_Bits.Ready;
   #HEAD_BUSY := #PLC_IN_Bits.Busy;
   #SYSTEM_RUN := #PLC_IN_Bits.Run;
   #CMD_COMPLETE := #PLC_IN_Bits.CommandCompleteFlag;



   // Bytes
   #ACTIVE_PRG := #PLC_IN_Bytes.CurrentPrgNumber;
END_REGION
END_FUNCTION_BLOCK

FUNCTION_BLOCK "MeasTable_SQ"   // FB15, GRAPH
AUTHOR : an38503
VERSION : 0.1
// stored: AcknowledgeErrorsRequired true, AutoNumber true, GraphVersion 6.0, InitialValuesAcquisition false, IsIECCheckEnabled false, LanguageInNetworks FBD, LockOperatingMode false, PermanentILProcessingInMANMode false, SetENOAutomatically false, SkipSteps false, UDAEnableTagReadback false, WithAlarmHandling true
   // inherited from GRAPH_BASE
   VAR
      OFF_SQ_BASE : Bool;
   END_VAR
   VAR_INPUT
      OFF_SQ { ExternalAccessible := 'False'; ExternalVisible := 'False'; ExternalWritable := 'False'} : Bool := false;   // Kette ausschalten
      INIT_SQ { ExternalAccessible := 'False'; ExternalVisible := 'False'; ExternalWritable := 'False'} : Bool := false;   // Kette in Initialzustand versetzen
      ACK_EF { ExternalAccessible := 'False'; ExternalVisible := 'False'; ExternalWritable := 'False'} : Bool := false;   // Alle Fehler und Störungen quittieren
      S_PREV { ExternalAccessible := 'False'; ExternalVisible := 'False'; ExternalWritable := 'False'} : Bool := false;   // Vorherigen Schritt am Parameter S_NO ausgeben
      S_NEXT { ExternalAccessible := 'False'; ExternalVisible := 'False'; ExternalWritable := 'False'} : Bool := false;   // Nächsten Schritt am Parameter S_NO anzeigen
      SW_AUTO { ExternalAccessible := 'False'; ExternalVisible := 'False'; ExternalWritable := 'False'} : Bool := false;   // Automatischer Betrieb
      SW_TAP { ExternalAccessible := 'False'; ExternalVisible := 'False'; ExternalWritable := 'False'} : Bool := false;   // Halbautomatisch/Weiterschalten mit Transition
      SW_TOP { ExternalAccessible := 'False'; ExternalVisible := 'False'; ExternalWritable := 'False'} : Bool := false;   // Halbautomatisch/Ignoriere Transition
      SW_MAN { ExternalAccessible := 'False'; ExternalVisible := 'False'; ExternalWritable := 'False'} : Bool := false;   // Handbetrieb
      S_SEL { ExternalAccessible := 'False'; ExternalVisible := 'False'; ExternalWritable := 'False'} : Int := 0;   // Schritt auswählen, der an S_NO ausgegeben werden soll
      S_ON { ExternalAccessible := 'False'; ExternalVisible := 'False'; ExternalWritable := 'False'} : Bool := false;   // Schritt aktivieren, der an Parameter S_NO anliegt
      S_OFF { ExternalAccessible := 'False'; ExternalVisible := 'False'; ExternalWritable := 'False'} : Bool := false;   // Schritt deaktivieren, der an Parameter S_NO anliegt
      T_PUSH { ExternalAccessible := 'False'; ExternalVisible := 'False'; ExternalWritable := 'False'} : Bool := false;   // Schaltfreigabe für Transition im halbautomatischen Betrieb
   END_VAR
   VAR_OUTPUT
      S_NO { ExternalAccessible := 'False'; ExternalVisible := 'False'; ExternalWritable := 'False'} : Int := 0;   // Schrittnummer
      S_MORE { ExternalAccessible := 'False'; ExternalVisible := 'False'; ExternalWritable := 'False'} : Bool := false;   // Weitere Schritte sind vorhanden und können in S_NO angezeigt werden.
      S_ACTIVE { ExternalAccessible := 'False'; ExternalVisible := 'False'; ExternalWritable := 'False'} : Bool := false;   // Schritt, der an Parameter S_NO angezeigt wird, ist aktiv
      ERR_FLT { ExternalAccessible := 'False'; ExternalVisible := 'False'; ExternalWritable := 'False'} : Bool := false;   // Sammelfehler Interlock oder Supervision
      AUTO_ON { ExternalAccessible := 'False'; ExternalVisible := 'False'; ExternalWritable := 'False'} : Bool := false;   // Automatischer Betrieb eingeschaltet
      TAP_ON { ExternalAccessible := 'False'; ExternalVisible := 'False'; ExternalWritable := 'False'} : Bool := false;   // Halbautomatischer Betrieb/Schritt mit Transition eingeschaltet
      TOP_ON { ExternalAccessible := 'False'; ExternalVisible := 'False'; ExternalWritable := 'False'} : Bool := false;   // Halbautomatischer Betrieb/Ignoriere Transition eingeschaltet
      MAN_ON { ExternalAccessible := 'False'; ExternalVisible := 'False'; ExternalWritable := 'False'} : Bool := false;   // Handbetrieb eingeschaltet
   END_VAR
   VAR
      SQ_ProgramRequest { S7_SetPoint := 'True'} : Bool;
      DataHasRead_1 : Bool;
   END_VAR
BEGIN
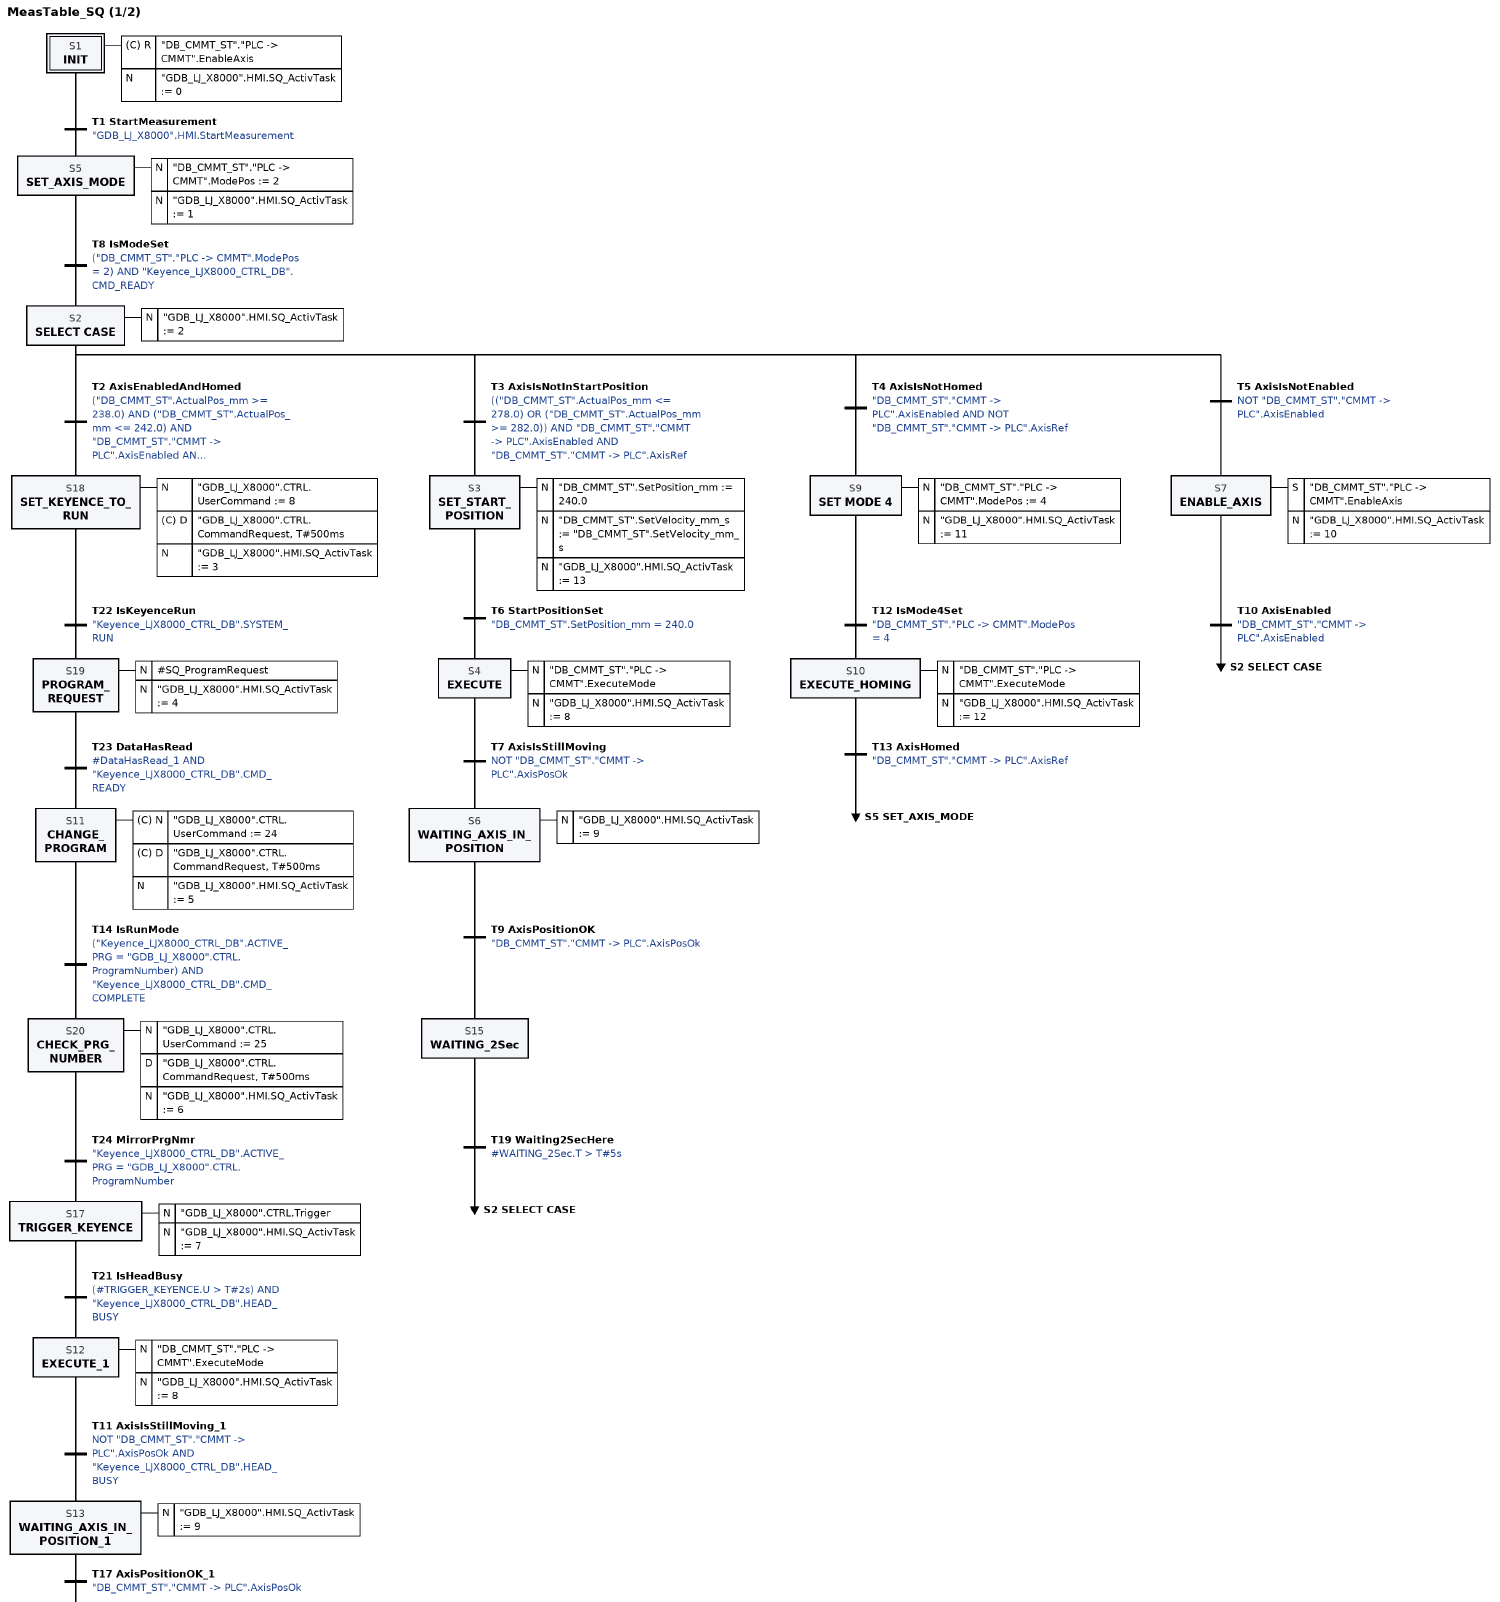
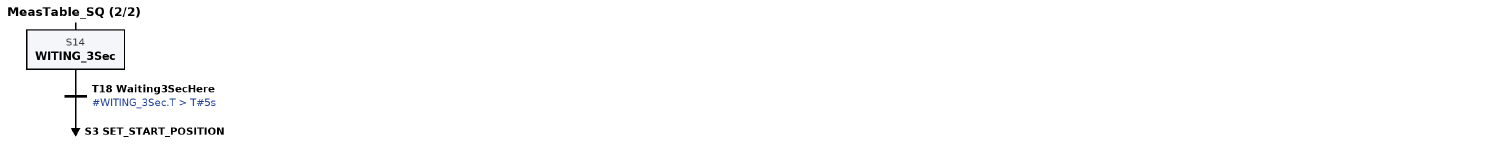
   // sequencer 1
   INITIAL_STEP INIT:   // S1, max time T#10S, warning time T#7S
      interlock C := "GDB_LJ_X8000".HMI.MeasurementMode AND NOT "GDB_LJ_X8000".HMI.HandMode;
      (C)     R    "DB_CMMT_ST"."PLC -> CMMT".EnableAxis
              N    "GDB_LJ_X8000".HMI.SQ_ActivTask := 0
   END_STEP
   TRANSITION StartMeasurement FROM INIT TO SET_AXIS_MODE   // T1
      := "GDB_LJ_X8000".HMI.StartMeasurement;
   END_TRANSITION
   STEP "SELECT CASE":   // S2, max time T#10S, warning time T#7S
              N    "GDB_LJ_X8000".HMI.SQ_ActivTask := 2
   END_STEP
   TRANSITION AxisEnabledAndHomed FROM "SELECT CASE" TO SET_KEYENCE_TO_RUN   // T2
      := ("DB_CMMT_ST".ActualPos_mm >= 238.0) AND ("DB_CMMT_ST".ActualPos_mm <= 242.0) AND "DB_CMMT_ST"."CMMT -> PLC".AxisEnabled AND "DB_CMMT_ST"."CMMT -> PLC".AxisRef AND "Keyence_LJX8000_CTRL_DB".CMD_READY;
   END_TRANSITION
   TRANSITION AxisIsNotInStartPosition FROM "SELECT CASE" TO SET_START_POSITION   // T3
      := (("DB_CMMT_ST".ActualPos_mm <= 278.0) OR ("DB_CMMT_ST".ActualPos_mm >= 282.0)) AND "DB_CMMT_ST"."CMMT -> PLC".AxisEnabled AND "DB_CMMT_ST"."CMMT -> PLC".AxisRef;
   END_TRANSITION
   TRANSITION AxisIsNotHomed FROM "SELECT CASE" TO "SET MODE 4"   // T4
      := "DB_CMMT_ST"."CMMT -> PLC".AxisEnabled AND NOT "DB_CMMT_ST"."CMMT -> PLC".AxisRef;
   END_TRANSITION
   TRANSITION AxisIsNotEnabled FROM "SELECT CASE" TO ENABLE_AXIS   // T5
      := NOT "DB_CMMT_ST"."CMMT -> PLC".AxisEnabled;
   END_TRANSITION
   STEP SET_START_POSITION:   // S3, max time T#10S, warning time T#7S
              N    "DB_CMMT_ST".SetPosition_mm := 240.0
              N    "DB_CMMT_ST".SetVelocity_mm_s := "DB_CMMT_ST".SetVelocity_mm_s
              N    "GDB_LJ_X8000".HMI.SQ_ActivTask := 13
   END_STEP
   TRANSITION StartPositionSet FROM SET_START_POSITION TO EXECUTE   // T6
      := "DB_CMMT_ST".SetPosition_mm = 240.0;
   END_TRANSITION
   STEP EXECUTE:   // S4, max time T#10S, warning time T#7S
              N    "DB_CMMT_ST"."PLC -> CMMT".ExecuteMode
              N    "GDB_LJ_X8000".HMI.SQ_ActivTask := 8
   END_STEP
   TRANSITION AxisIsStillMoving FROM EXECUTE TO WAITING_AXIS_IN_POSITION   // T7
      := NOT "DB_CMMT_ST"."CMMT -> PLC".AxisPosOk;
   END_TRANSITION
   STEP SET_AXIS_MODE:   // S5, max time T#10S, warning time T#7S
              N    "DB_CMMT_ST"."PLC -> CMMT".ModePos := 2
              N    "GDB_LJ_X8000".HMI.SQ_ActivTask := 1
   END_STEP
   TRANSITION IsModeSet FROM SET_AXIS_MODE TO "SELECT CASE"   // T8
      := ("DB_CMMT_ST"."PLC -> CMMT".ModePos = 2) AND "Keyence_LJX8000_CTRL_DB".CMD_READY;
   END_TRANSITION
   STEP WAITING_AXIS_IN_POSITION:   // S6, max time T#10S, warning time T#7S
              N    "GDB_LJ_X8000".HMI.SQ_ActivTask := 9
   END_STEP
   TRANSITION AxisPositionOK FROM WAITING_AXIS_IN_POSITION TO WAITING_2Sec   // T9
      := "DB_CMMT_ST"."CMMT -> PLC".AxisPosOk;
   END_TRANSITION
   STEP ENABLE_AXIS:   // S7, max time T#10S, warning time T#7S
              S    "DB_CMMT_ST"."PLC -> CMMT".EnableAxis
              N    "GDB_LJ_X8000".HMI.SQ_ActivTask := 10
   END_STEP
   TRANSITION AxisEnabled FROM ENABLE_AXIS TO "SELECT CASE"   // T10, jump
      := "DB_CMMT_ST"."CMMT -> PLC".AxisEnabled;
   END_TRANSITION
   STEP "SET MODE 4":   // S9, max time T#10S, warning time T#7S
              N    "DB_CMMT_ST"."PLC -> CMMT".ModePos := 4
              N    "GDB_LJ_X8000".HMI.SQ_ActivTask := 11
   END_STEP
   TRANSITION IsMode4Set FROM "SET MODE 4" TO EXECUTE_HOMING   // T12
      := "DB_CMMT_ST"."PLC -> CMMT".ModePos = 4;
   END_TRANSITION
   STEP EXECUTE_HOMING:   // S10, max time T#10S, warning time T#7S
              N    "DB_CMMT_ST"."PLC -> CMMT".ExecuteMode
              N    "GDB_LJ_X8000".HMI.SQ_ActivTask := 12
   END_STEP
   TRANSITION AxisHomed FROM EXECUTE_HOMING TO SET_AXIS_MODE   // T13, jump
      := "DB_CMMT_ST"."CMMT -> PLC".AxisRef;
   END_TRANSITION
   STEP CHANGE_PROGRAM:   // S11, max time T#10S, warning time T#7S
      (C)     N    "GDB_LJ_X8000".CTRL.UserCommand := 24
      (C)     D    "GDB_LJ_X8000".CTRL.CommandRequest, T#500ms
              N    "GDB_LJ_X8000".HMI.SQ_ActivTask := 5
   END_STEP
   TRANSITION IsRunMode FROM CHANGE_PROGRAM TO CHECK_PRG_NUMBER   // T14
      := ("Keyence_LJX8000_CTRL_DB".ACTIVE_PRG = "GDB_LJ_X8000".CTRL.ProgramNumber) AND "Keyence_LJX8000_CTRL_DB".CMD_COMPLETE;
   END_TRANSITION
   STEP TRIGGER_KEYENCE:   // S17, max time T#10S, warning time T#7S
              N    "GDB_LJ_X8000".CTRL.Trigger
              N    "GDB_LJ_X8000".HMI.SQ_ActivTask := 7
   END_STEP
   TRANSITION IsHeadBusy FROM TRIGGER_KEYENCE TO EXECUTE_1   // T21
      := (#TRIGGER_KEYENCE.U > T#2s) AND "Keyence_LJX8000_CTRL_DB".HEAD_BUSY;
   END_TRANSITION
   STEP EXECUTE_1:   // S12, max time T#10S, warning time T#7S
              N    "DB_CMMT_ST"."PLC -> CMMT".ExecuteMode
              N    "GDB_LJ_X8000".HMI.SQ_ActivTask := 8
   END_STEP
   TRANSITION AxisIsStillMoving_1 FROM EXECUTE_1 TO WAITING_AXIS_IN_POSITION_1   // T11
      := NOT "DB_CMMT_ST"."CMMT -> PLC".AxisPosOk AND "Keyence_LJX8000_CTRL_DB".HEAD_BUSY;
   END_TRANSITION
   STEP WITING_3Sec:   // S14, max time T#10S, warning time T#7S
   END_STEP
   TRANSITION Waiting3SecHere FROM WITING_3Sec TO SET_START_POSITION   // T18, jump
      := #WITING_3Sec.T > T#5s;
   END_TRANSITION
   STEP WAITING_AXIS_IN_POSITION_1:   // S13, max time T#10S, warning time T#7S
              N    "GDB_LJ_X8000".HMI.SQ_ActivTask := 9
   END_STEP
   TRANSITION AxisPositionOK_1 FROM WAITING_AXIS_IN_POSITION_1 TO WITING_3Sec   // T17
      := "DB_CMMT_ST"."CMMT -> PLC".AxisPosOk;
   END_TRANSITION
   STEP WAITING_2Sec:   // S15, max time T#10S, warning time T#7S
   END_STEP
   TRANSITION Waiting2SecHere FROM WAITING_2Sec TO "SELECT CASE"   // T19, jump
      := #WAITING_2Sec.T > T#5s;
   END_TRANSITION
   STEP SET_KEYENCE_TO_RUN:   // S18, max time T#10S, warning time T#7S
      interlock C := NOT "Keyence_LJX8000_CTRL_DB".SYSTEM_RUN;
              N    "GDB_LJ_X8000".CTRL.UserCommand := 8
      (C)     D    "GDB_LJ_X8000".CTRL.CommandRequest, T#500ms
              N    "GDB_LJ_X8000".HMI.SQ_ActivTask := 3
   END_STEP
   TRANSITION IsKeyenceRun FROM SET_KEYENCE_TO_RUN TO PROGRAM_REQUEST   // T22
      := "Keyence_LJX8000_CTRL_DB".SYSTEM_RUN;
   END_TRANSITION
   STEP PROGRAM_REQUEST:   // S19, max time T#10S, warning time T#7S
              N    #SQ_ProgramRequest
              N    "GDB_LJ_X8000".HMI.SQ_ActivTask := 4
   END_STEP
   TRANSITION DataHasRead FROM PROGRAM_REQUEST TO CHANGE_PROGRAM   // T23
      := #DataHasRead_1 AND "Keyence_LJX8000_CTRL_DB".CMD_READY;
   END_TRANSITION
   STEP CHECK_PRG_NUMBER:   // S20, max time T#10S, warning time T#7S
              N    "GDB_LJ_X8000".CTRL.UserCommand := 25
              D    "GDB_LJ_X8000".CTRL.CommandRequest, T#500ms
              N    "GDB_LJ_X8000".HMI.SQ_ActivTask := 6
   END_STEP
   TRANSITION MirrorPrgNmr FROM CHECK_PRG_NUMBER TO TRIGGER_KEYENCE   // T24
      := "Keyence_LJX8000_CTRL_DB".ACTIVE_PRG = "GDB_LJ_X8000".CTRL.ProgramNumber;
   END_TRANSITION
END_FUNCTION_BLOCK

FUNCTION_BLOCK "B.01813_SIPP"   // FB7, LAD
{ S7_Optimized_Access := 'TRUE' }
VERSION : 0.1
// stored: AutoNumber true, IsIECCheckEnabled false, IsRetainMemResEnabled false, MemoryReserve 100, SetENOAutomatically false, UDAEnableTagReadback false
   VAR
      SQ_Activation_Time : UDInt;
      SQ_Act_time_inH : Real;
   END_VAR
BEGIN

REGION Network 1
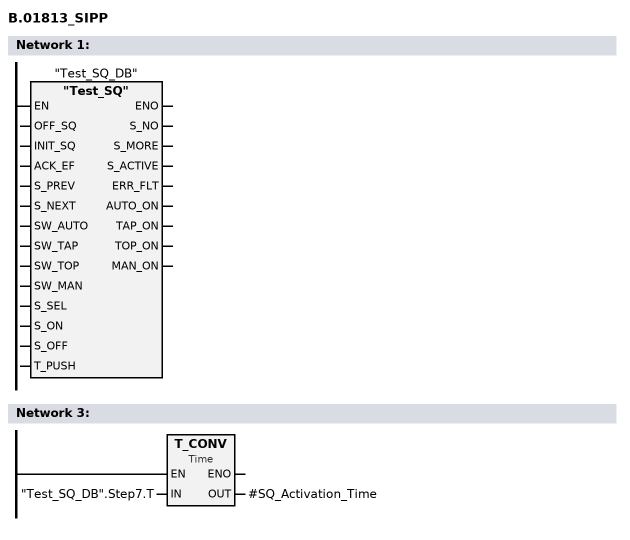
   RUNG wire#powerrail
      "Test_SQ_DB"(OFF_SQ :=, INIT_SQ :=, ACK_EF :=, S_PREV :=, S_NEXT :=, SW_AUTO :=, SW_TAP :=, SW_TOP :=, SW_MAN :=, S_SEL :=, S_ON :=, S_OFF :=, T_PUSH :=, S_NO =>, S_MORE =>, S_ACTIVE =>, ERR_FLT =>, AUTO_ON =>, TAP_ON =>, TOP_ON =>, MAN_ON =>)
   END_RUNG
   // the same network as SCL:
   "Test_SQ_DB"();   // "Test_SQ"
END_REGION

REGION Network 2 (SCL)
   #SQ_Act_time_inH := #SQ_Activation_Time / 1000.0 / 60 / 60;
END_REGION

REGION Network 3
   RUNG wire#powerrail
      { S7_Templates := "[src_type := Time, dest_type := UDInt]" } T_CONV(IN := "Test_SQ_DB".Step7.T, OUT => #SQ_Activation_Time)
   END_RUNG
   // the same network as SCL:
   T_CONV(IN := "Test_SQ_DB".Step7.T, OUT => #SQ_Activation_Time);
END_REGION
END_FUNCTION_BLOCK

FUNCTION_BLOCK "Test_SQ"   // FB8, GRAPH
VERSION : 0.1
// stored: AcknowledgeErrorsRequired true, AutoNumber true, GraphVersion 6.0, InitialValuesAcquisition false, IsIECCheckEnabled false, LanguageInNetworks FBD, LockOperatingMode false, PermanentILProcessingInMANMode false, SetENOAutomatically false, SkipSteps false, UDAEnableTagReadback false, WithAlarmHandling true
   // inherited from GRAPH_BASE
   VAR
      OFF_SQ_BASE : Bool;
   END_VAR
   VAR_INPUT
      OFF_SQ { ExternalAccessible := 'False'; ExternalVisible := 'False'; ExternalWritable := 'False'} : Bool := false;   // Kette ausschalten
      INIT_SQ { ExternalAccessible := 'False'; ExternalVisible := 'False'; ExternalWritable := 'False'} : Bool := false;   // Kette in Initialzustand versetzen
      ACK_EF { ExternalAccessible := 'False'; ExternalVisible := 'False'; ExternalWritable := 'False'} : Bool := false;   // Alle Fehler und Störungen quittieren
      S_PREV { ExternalAccessible := 'False'; ExternalVisible := 'False'; ExternalWritable := 'False'} : Bool := false;   // Vorherigen Schritt am Parameter S_NO ausgeben
      S_NEXT { ExternalAccessible := 'False'; ExternalVisible := 'False'; ExternalWritable := 'False'} : Bool := false;   // Nächsten Schritt am Parameter S_NO anzeigen
      SW_AUTO { ExternalAccessible := 'False'; ExternalVisible := 'False'; ExternalWritable := 'False'} : Bool := false;   // Automatischer Betrieb
      SW_TAP { ExternalAccessible := 'False'; ExternalVisible := 'False'; ExternalWritable := 'False'} : Bool := false;   // Halbautomatisch/Weiterschalten mit Transition
      SW_TOP { ExternalAccessible := 'False'; ExternalVisible := 'False'; ExternalWritable := 'False'} : Bool := false;   // Halbautomatisch/Ignoriere Transition
      SW_MAN { ExternalAccessible := 'False'; ExternalVisible := 'False'; ExternalWritable := 'False'} : Bool := false;   // Handbetrieb
      S_SEL { ExternalAccessible := 'False'; ExternalVisible := 'False'; ExternalWritable := 'False'} : Int := 0;   // Schritt auswählen, der an S_NO ausgegeben werden soll
      S_ON { ExternalAccessible := 'False'; ExternalVisible := 'False'; ExternalWritable := 'False'} : Bool := false;   // Schritt aktivieren, der an Parameter S_NO anliegt
      S_OFF { ExternalAccessible := 'False'; ExternalVisible := 'False'; ExternalWritable := 'False'} : Bool := false;   // Schritt deaktivieren, der an Parameter S_NO anliegt
      T_PUSH { ExternalAccessible := 'False'; ExternalVisible := 'False'; ExternalWritable := 'False'} : Bool := false;   // Schaltfreigabe für Transition im halbautomatischen Betrieb
   END_VAR
   VAR_OUTPUT
      S_NO { ExternalAccessible := 'False'; ExternalVisible := 'False'; ExternalWritable := 'False'} : Int := 0;   // Schrittnummer
      S_MORE { ExternalAccessible := 'False'; ExternalVisible := 'False'; ExternalWritable := 'False'} : Bool := false;   // Weitere Schritte sind vorhanden und können in S_NO angezeigt werden.
      S_ACTIVE { ExternalAccessible := 'False'; ExternalVisible := 'False'; ExternalWritable := 'False'} : Bool := false;   // Schritt, der an Parameter S_NO angezeigt wird, ist aktiv
      ERR_FLT { ExternalAccessible := 'False'; ExternalVisible := 'False'; ExternalWritable := 'False'} : Bool := false;   // Sammelfehler Interlock oder Supervision
      AUTO_ON { ExternalAccessible := 'False'; ExternalVisible := 'False'; ExternalWritable := 'False'} : Bool := false;   // Automatischer Betrieb eingeschaltet
      TAP_ON { ExternalAccessible := 'False'; ExternalVisible := 'False'; ExternalWritable := 'False'} : Bool := false;   // Halbautomatischer Betrieb/Schritt mit Transition eingeschaltet
      TOP_ON { ExternalAccessible := 'False'; ExternalVisible := 'False'; ExternalWritable := 'False'} : Bool := false;   // Halbautomatischer Betrieb/Ignoriere Transition eingeschaltet
      MAN_ON { ExternalAccessible := 'False'; ExternalVisible := 'False'; ExternalWritable := 'False'} : Bool := false;   // Handbetrieb eingeschaltet
   END_VAR
BEGIN
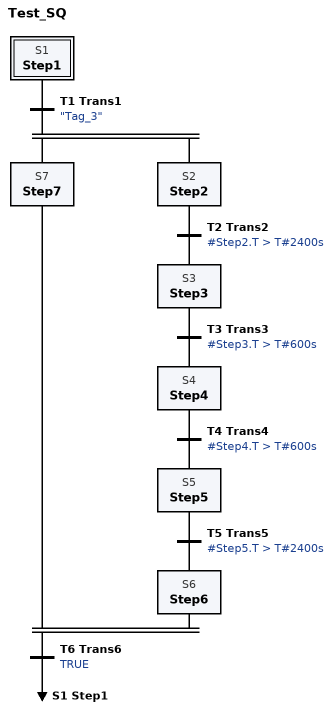
   // sequencer 1
   INITIAL_STEP Step1:   // S1, max time T#10S, warning time T#7S
   END_STEP
   TRANSITION Trans1 FROM Step1 TO (Step7, Step2)   // T1
      := "Tag_3";
   END_TRANSITION
   STEP Step2:   // S2, max time T#10S, warning time T#7S
   END_STEP
   TRANSITION Trans2 FROM Step2 TO Step3   // T2
      := #Step2.T > T#2400s;
   END_TRANSITION
   STEP Step3:   // S3, max time T#10S, warning time T#7S
   END_STEP
   TRANSITION Trans3 FROM Step3 TO Step4   // T3
      := #Step3.T > T#600s;
   END_TRANSITION
   STEP Step4:   // S4, max time T#10S, warning time T#7S
   END_STEP
   TRANSITION Trans4 FROM Step4 TO Step5   // T4
      := #Step4.T > T#600s;
   END_TRANSITION
   STEP Step5:   // S5, max time T#10S, warning time T#7S
   END_STEP
   TRANSITION Trans5 FROM Step5 TO Step6   // T5
      := #Step5.T > T#2400s;
   END_TRANSITION
   STEP Step6:   // S6, max time T#10S, warning time T#7S
   END_STEP
   STEP Step7:   // S7, max time T#10S, warning time T#7S
   END_STEP
   TRANSITION Trans6 FROM (Step6, Step7) TO Step1   // T6, jump
      := TRUE;
   END_TRANSITION
END_FUNCTION_BLOCK

FUNCTION_BLOCK "FB_DATA_LOGGING"   // FB13, LAD
{ S7_Optimized_Access := 'TRUE' }
VERSION : 0.1
// stored: AutoNumber true, IsIECCheckEnabled false, IsRetainMemResEnabled false, MemoryReserve 100, SetENOAutomatically false, UDAEnableTagReadback false
   VAR
      DataLogCreate_Instance { S7_SetPoint := 'True'} : DataLogCreate;
      DataLogWrite_Instance { S7_SetPoint := 'True'} : DataLogWrite;
      DataLogNewFile_Instance { S7_SetPoint := 'True'} : DataLogNewFile;
      DataLogNewFile_Instance_1 { S7_SetPoint := 'True'} : DataLogNewFile;
      DataLogDelete_Instance { S7_SetPoint := 'True'} : DataLogDelete;
      DataLogClear_Instance { S7_SetPoint := 'True'} : DataLogClear;
   END_VAR
BEGIN

REGION Network 1: Data Log Create
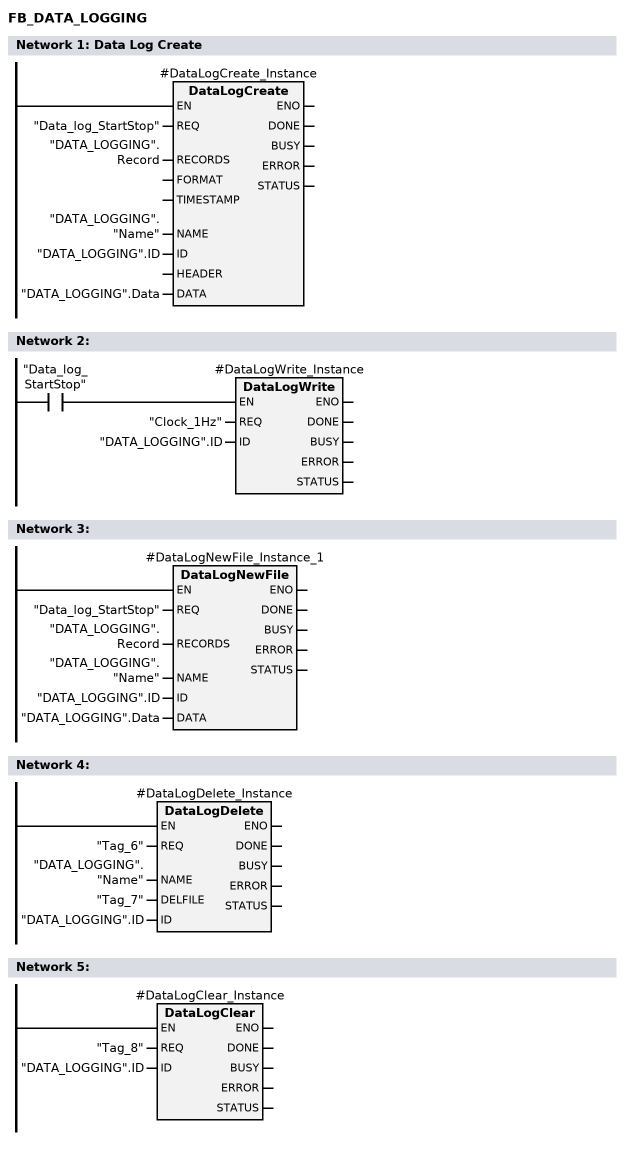
   RUNG wire#powerrail
      #DataLogCreate_Instance.DataLogCreate(REQ := "Data_log_StartStop", RECORDS := "DATA_LOGGING".Record, FORMAT :=, TIMESTAMP :=, "NAME" := "DATA_LOGGING"."Name", ID := "DATA_LOGGING".ID, HEADER :=, DATA := "DATA_LOGGING".Data, DONE =>, BUSY =>, ERROR =>, STATUS =>)
   END_RUNG
   // the same network as SCL:
   #DataLogCreate_Instance(REQ := "Data_log_StartStop",   // DataLogCreate
                           RECORDS := "DATA_LOGGING".Record,
                           "NAME" := "DATA_LOGGING"."Name",
                           ID := "DATA_LOGGING".ID,
                           DATA := "DATA_LOGGING".Data);
END_REGION

REGION Network 2
   RUNG wire#powerrail
      Contact( "Data_log_StartStop" )
      #DataLogWrite_Instance.DataLogWrite(REQ := "Clock_1Hz", ID := "DATA_LOGGING".ID, DONE =>, BUSY =>, ERROR =>, STATUS =>)
   END_RUNG
   // the same network as SCL:
   IF "Data_log_StartStop" THEN
       #DataLogWrite_Instance(REQ := "Clock_1Hz", ID := "DATA_LOGGING".ID);   // DataLogWrite
   END_IF;
END_REGION

REGION Network 3
   RUNG wire#powerrail
      { S7_Templates := "card := 1" } #DataLogNewFile_Instance_1.DataLogNewFile(REQ := "Data_log_StartStop", RECORDS := "DATA_LOGGING".Record, "NAME" := "DATA_LOGGING"."Name", ID := "DATA_LOGGING".ID, Data := "DATA_LOGGING".Data, DONE =>, BUSY =>, ERROR =>, STATUS =>)
   END_RUNG
   // the same network as SCL:
   #DataLogNewFile_Instance_1(REQ := "Data_log_StartStop",   // DataLogNewFile
                           RECORDS := "DATA_LOGGING".Record,
                           "NAME" := "DATA_LOGGING"."Name",
                           ID := "DATA_LOGGING".ID,
                           Data := "DATA_LOGGING".Data);
END_REGION

REGION Network 4
   RUNG wire#powerrail
      #DataLogDelete_Instance.DataLogDelete(REQ := "Tag_6", "NAME" := "DATA_LOGGING"."Name", DelFile := "Tag_7", ID := "DATA_LOGGING".ID, DONE =>, BUSY =>, ERROR =>, STATUS =>)
   END_RUNG
   // the same network as SCL:
   #DataLogDelete_Instance(REQ := "Tag_6",   // DataLogDelete
                           "NAME" := "DATA_LOGGING"."Name",
                           DelFile := "Tag_7",
                           ID := "DATA_LOGGING".ID);
END_REGION

REGION Network 5
   RUNG wire#powerrail
      #DataLogClear_Instance.DataLogClear(REQ := "Tag_8", ID := "DATA_LOGGING".ID, DONE =>, BUSY =>, ERROR =>, STATUS =>)
   END_RUNG
   // the same network as SCL:
   #DataLogClear_Instance(REQ := "Tag_8", ID := "DATA_LOGGING".ID);   // DataLogClear
END_REGION
END_FUNCTION_BLOCK

FUNCTION_BLOCK "Main_Safety_RTG1"   // FB1, F_FBD
{ S7_Optimized_Access := 'TRUE' }
VERSION : 0.1
// stored: AutoNumber false, IsIECCheckEnabled false, UDAEnableTagReadback false
BEGIN
END_FUNCTION_BLOCK

FUNCTION "Baustein_1" : Void   // FC3, FBD
{ S7_Optimized_Access := 'TRUE' }
VERSION : 0.1
// stored: AutoNumber true, IsIECCheckEnabled false, SetENOAutomatically false, UDAEnableTagReadback false
BEGIN

REGION Network 1
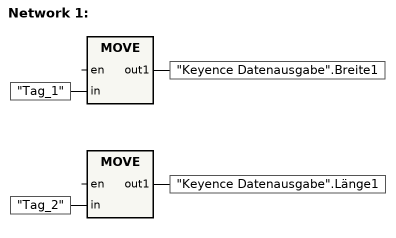
   "Keyence Datenausgabe".Breite1 := "Tag_1";
   "Keyence Datenausgabe".Länge1 := "Tag_2";
END_REGION
END_FUNCTION

FUNCTION "FC_TransferDataPLC_LJX8000" : Void   // FC4, LAD
{ S7_Optimized_Access := 'TRUE' }
VERSION : 0.1
// stored: AutoNumber true, IsIECCheckEnabled false, SetENOAutomatically false, UDAEnableTagReadback false
BEGIN

REGION Network 1: PLC to LJ_X8000 bits
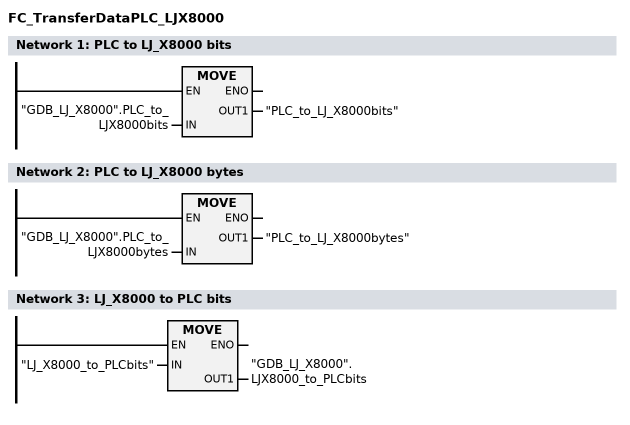
   RUNG wire#powerrail
      Move(in := "GDB_LJ_X8000".PLC_to_LJX8000bits, out1 => "PLC_to_LJ_X8000bits")
   END_RUNG
   // the same network as SCL:
   "PLC_to_LJ_X8000bits" := "GDB_LJ_X8000".PLC_to_LJX8000bits;
END_REGION

REGION Network 2: PLC to LJ_X8000 bytes
   RUNG wire#powerrail
      Move(in := "GDB_LJ_X8000".PLC_to_LJX8000bytes, out1 => "PLC_to_LJ_X8000bytes")
   END_RUNG
   // the same network as SCL:
   "PLC_to_LJ_X8000bytes" := "GDB_LJ_X8000".PLC_to_LJX8000bytes;
END_REGION

REGION Network 3: LJ_X8000 to PLC bits
   RUNG wire#powerrail
      Move(in := "LJ_X8000_to_PLCbits", out1 => "GDB_LJ_X8000".LJX8000_to_PLCbits)
   END_RUNG
   // the same network as SCL:
   "GDB_LJ_X8000".LJX8000_to_PLCbits := "LJ_X8000_to_PLCbits";
END_REGION
END_FUNCTION

FUNCTION_BLOCK "LJ_X8000_CTRL"   // FB12, LAD
{ S7_Optimized_Access := 'TRUE' }
VERSION : 0.1
// stored: AutoNumber true, IsIECCheckEnabled false, IsRetainMemResEnabled false, MemoryReserve 100, SetENOAutomatically false, UDAEnableTagReadback false
BEGIN
END_FUNCTION_BLOCK

DATA_BLOCK "Main_Safety_RTG1_DB"   // DB1, F_DB
NAME : FUSI
VERSION : 0.1
// stored: AutoNumber true, DBAccessibleFromOPCUA true, DBAccessibleFromWebserver true, InstanceOfName Main_Safety_RTG1, InstanceOfType FB
"Main_Safety_RTG1"
BEGIN
END_DATA_BLOCK

DATA_BLOCK "FB_Database_DB"   // DB9
VERSION : 0.1
// stored: AutoNumber true, DBAccessibleFromOPCUA true, DBAccessibleFromWebserver true, InstanceOfName FB_Database, InstanceOfType FB
"FB_Database"
BEGIN
END_DATA_BLOCK

DATA_BLOCK "FB_DATA_LOGGING_DB"   // DB26
VERSION : 0.1
// stored: AutoNumber true, DBAccessibleFromOPCUA true, DBAccessibleFromWebserver true, InstanceOfName FB_DATA_LOGGING, InstanceOfType FB
"FB_DATA_LOGGING"
BEGIN
END_DATA_BLOCK

DATA_BLOCK "FFT_BREMEN_SPS_Connection_DB_2"   // DB38
{ S7_Optimized_Access := 'TRUE' }
// stored: AutoNumber true, DBAccessibleFromOPCUA true, DBAccessibleFromWebserver true, InstanceOfName TCON_IP_v4, OfSystemLibElement TCON_IP_v4, OfSystemLibVersion 1.0
"TCON_IP_v4"
   // VAR
   //    InterfaceId : HW_ANY := 64;
   //    ID : CONN_OUC := 3;
   //    ConnectionType : Byte;
   //    ActiveEstablished : Bool := true;
   //    RemoteAddress { S7_SetPoint := 'True'} : IP_V4;
   //    RemotePort : UInt := 2001;
   //    LocalPort : UInt := 2000;
   // END_VAR
BEGIN
   RemoteAddress.ADDR[1] := 10;
   RemoteAddress.ADDR[2] := 183;
   RemoteAddress.ADDR[3] := 122;
   RemoteAddress.ADDR[4] := 3;
END_DATA_BLOCK

DATA_BLOCK "F_TRIG_DB"   // DB23
// stored: AutoNumber true, DBAccessibleFromOPCUA true, DBAccessibleFromWebserver true, InstanceOfName F_TRIG, OfSystemLibElement F_TRIG, OfSystemLibVersion 1.0
"F_TRIG"
   // VAR_INPUT
   //    CLK : Bool;
   // END_VAR
   // VAR_OUTPUT
   //    Q : Bool;
   // END_VAR
   // VAR
   //    Stat_Bit : Bool;
   // END_VAR
BEGIN
END_DATA_BLOCK

DATA_BLOCK "IEC_Timer_0_DB"   // DB22
{ S7_Optimized_Access := 'TRUE' }
// stored: AutoNumber true, DBAccessibleFromOPCUA true, DBAccessibleFromWebserver true, InstanceOfName IEC_TIMER, OfSystemLibElement IEC_TIMER, OfSystemLibVersion 1.0
"IEC_TIMER"
   // VAR
   //    PT : Time;
   //    ET { ExternalWritable := 'False'} : Time;
   //    IN : Bool;
   //    Q { ExternalWritable := 'False'} : Bool;
   // END_VAR
BEGIN
END_DATA_BLOCK

DATA_BLOCK "R_TRIG_DB"   // DB19
// stored: AutoNumber true, DBAccessibleFromOPCUA true, DBAccessibleFromWebserver true, InstanceOfName R_TRIG, OfSystemLibElement R_TRIG, OfSystemLibVersion 1.0
"R_TRIG"
   // VAR_INPUT
   //    CLK : Bool;
   // END_VAR
   // VAR_OUTPUT
   //    Q : Bool;
   // END_VAR
   // VAR
   //    Stat_Bit : Bool;
   // END_VAR
BEGIN
END_DATA_BLOCK

DATA_BLOCK "B.01813_SIPP_DB"   // DB20
VERSION : 0.1
// stored: AutoNumber true, DBAccessibleFromOPCUA true, DBAccessibleFromWebserver true, InstanceOfName B.01813_SIPP, InstanceOfType FB
"B.01813_SIPP"
BEGIN
END_DATA_BLOCK

DATA_BLOCK "Test_SQ_DB"   // DB21
VERSION : 0.1
// stored: AutoNumber true, DBAccessibleFromOPCUA true, DBAccessibleFromWebserver true, InstanceOfName Test_SQ, InstanceOfType FB
"Test_SQ"
BEGIN
END_DATA_BLOCK

DATA_BLOCK "B.05847_FFB_DB"   // DB11
VERSION : 0.1
// stored: AutoNumber true, DBAccessibleFromOPCUA true, DBAccessibleFromWebserver true, InstanceOfName B.05847_FFB, InstanceOfType FB
"B.05847_FFB"
BEGIN
END_DATA_BLOCK

DATA_BLOCK "FB_LJ_X8000_CTRL_DB"   // DB24
VERSION : 0.1
// stored: AutoNumber true, DBAccessibleFromOPCUA true, DBAccessibleFromWebserver true, InstanceOfName FB_LJ_X8000, InstanceOfType FB
"FB_LJ_X8000"
BEGIN
END_DATA_BLOCK

DATA_BLOCK "Keyence_LJX8000_CTRL_DB"   // DB27
VERSION : 0.1
// stored: AutoNumber true, DBAccessibleFromOPCUA true, DBAccessibleFromWebserver true, InstanceOfName Keyence_LJX8000_CTRL, InstanceOfType FB
"Keyence_LJX8000_CTRL"
BEGIN
END_DATA_BLOCK

DATA_BLOCK "MeasTable_SQ_DB"   // DB28
AUTHOR : an38503
VERSION : 0.1
// stored: AutoNumber true, DBAccessibleFromOPCUA true, DBAccessibleFromWebserver true, InstanceOfName MeasTable_SQ, InstanceOfType FB
"MeasTable_SQ"
BEGIN
END_DATA_BLOCK

DATA_BLOCK "Gatewas_RS232_LK_G5000_DB"   // DB18
VERSION : 0.1
// stored: AutoNumber true, DBAccessibleFromOPCUA true, DBAccessibleFromWebserver true, InstanceOfName Gatewas_RS232_LK_G5000, InstanceOfType FB
"Gatewas_RS232_LK_G5000"
BEGIN
END_DATA_BLOCK

DATA_BLOCK "LK_G5000_DB"   // DB17
VERSION : 0.1
// stored: AutoNumber true, DBAccessibleFromOPCUA true, DBAccessibleFromWebserver true, InstanceOfName LK_G5000, InstanceOfType FB
"LK_G5000"
BEGIN
END_DATA_BLOCK

DATA_BLOCK "FESTO_CMMT_ST_DB"   // DB12
VERSION : 0.1
// stored: AutoNumber true, DBAccessibleFromOPCUA true, DBAccessibleFromWebserver true, InstanceOfName FESTO_CMMT_ST, InstanceOfType FB
"FESTO_CMMT_ST"
BEGIN
END_DATA_BLOCK

DATA_BLOCK "Festo_ClampingTorque_DB"   // DB15
AUTHOR : Festo SE & Co. KG
FAMILY : Drives
VERSION : 1.0
// stored: AutoNumber true, DBAccessibleFromOPCUA true, DBAccessibleFromWebserver true, InstanceOfName Festo_ClampingTorque, InstanceOfType FB
"Festo_ClampingTorque"
BEGIN
END_DATA_BLOCK
